FUNCTION_BLOCK FB_Analog_Out_Minimum
VAR_INPUT
	Minimum																: REAL;
END_VAR
VAR_IN_OUT
	Input1																: REAL;
	Input2																: REAL;
END_VAR
VAR
	Last1																: REAL	:= -1;
	Last2																: REAL	:= -1;
END_VAR

// Phase 0 - FB_Analog_Out_Minimum
// Rev 1.0 - April 3, 2024

IF Input2 <> Last2 THEN
	Input2																:= SEL(Input2 < Minimum, Input2, Minimum);
	Last2																:= Input2;
	Input1																:= Input2;
	Last1																:= Input2;
ELSIF Input1 <> Last1 THEN
	Input1																:= SEL(Input1 < Minimum, Input1, Minimum);
	Last1																:= Input1;
	Input2																:= Input1;
	Last2																:= Input1;
END_IF

END_FUNCTION_BLOCK

(* stored: Version 1.1.0.1, ProductVersion 3.1.4024.12
   POU FB_Analog_Out_Minimum: Id {732ebd4f-67ec-4dfe-b943-21f066cb8284}, SpecialFunc None *)
